VAR_GLOBAL
	// Define COM Ports/Buffers incl. library Tc2_SerialCom
	E1_SerialRXBuffer : ComBuffer;
	E1_SerialTXBuffer : ComBuffer;
	
	// Serial Terminal
	fbSerialLineControl_E1: SerialLineControl;

	//SERIAL IO
	E1_stComIn		AT %I*	:	EL6inData22B;
	E1_stComOut		AT %Q*	:	EL6outData22B;
	
	
	
	
	// Define COM Ports/Buffers incl. library Tc2_SerialCom
	E2_SerialRXBuffer : ComBuffer;
	E2_SerialTXBuffer : ComBuffer;
	
	// Serial Terminal
	fbSerialLineControl_E2: SerialLineControl;

	//SERIAL IO
	E2_stComIn		AT %I*	:	EL6inData22B;
	E2_stComOut		AT %Q*	:	EL6outData22B;
	
	
	
END_VAR

(* stored: Version 1.1.0.1, ProductVersion 3.1.4024.3
   GVL GVL_COM: Id {7c8ef01c-139d-4a9c-a18a-777693166eb4} *)
